// Brief: Slave Arm Adjust
FUNCTION_BLOCK PUBLIC FB_SlaveCtrlKineCaliSample EXTENDS FB_SlaveCtrlAdjust
VAR CONSTANT
	m_sampleNum :INT :=15;
END_VAR
VAR
	// sample joint position 
	m_sampleSetupJntPos :ARRAY[1..m_sampleNum] OF Vec5d;
	m_sampleSlaveJntPos :ARRAY[1..m_sampleNum] OF Vec6d;
	
	// sample signal
	m_sampleSignal : FB_AdjustLongPress;
	
	// current sample number
	m_curSampleNum :INT :=1;
	
	m_logStr:STRING;
	m_armStr:STRING;
	
END_VAR

// override this function in each exact controller
METHOD PROTECTED calcCmdJntPos : BOOL
VAR_IN_OUT CONSTANT
	i_endoscopePose : ST_Frame;
	i_masterStatus :ST_MasterStatus;
	i_setupStatus: ST_SetupStatus;
	i_slaveArm :FB_SlaveArm;
END_VAR
VAR
	i:INT;
END_VAR
SUPER^.calcCmdJntPos(i_endoscopePose,i_masterStatus, i_setupStatus, i_slaveArm);

IF m_curSampleNum > m_sampleNum THEN
	m_isFinished :=TRUE;
	AGILOG_DebugStop();
	RETURN;
END_IF
	
IF m_sampleSignal.run(i_slaveArm.m_adjustIO) THEN
	
	m_sampleSetupJntPos[m_curSampleNum] := SetupArmControl.m_setupRobot.m_setupArms[i_slaveArm.armIdx].curJntPos;
	m_sampleSlaveJntPos[m_curSampleNum] := i_slaveArm.curDHJntPos;
	
	AGILOG_DEBUG(m_armStr, FALSE, 1);
	
//	AGILOG_DEBUG(SetupArmControl.m_setupRobot.m_setupArms[i_slaveArm.armIdx].curJntPos, FALSE, 2);
//	AGILOG_DEBUG(i_slaveArm.curDHJntPos, FALSE, 1);
	
	AGILOG_DEBUG(RobotDynamics.m_instruViewCheck.m_instruPoseInScope[i_slaveArm.armIdx].m_pos,FALSE, 1);
	
	m_curSampleNum := m_curSampleNum +1;
END_IF
END_METHOD

METHOD PUBLIC Init : BOOL
VAR_IN_OUT CONSTANT
	i_slaveArm	:FB_SlaveArm;
END_VAR
VAR_IN_OUT 
	r_slaveArmCtrlCmd :ST_SlaveArmCtrlCmds;
END_VAR

VAR
	fileName:STRING;
END_VAR
//init
SUPER^.Init(i_slaveArm,r_slaveArmCtrlCmd);

m_curSampleNum:=1;
 
fileName := CONCAT('kineCaliSample_arm', INT_TO_STRING(i_slaveArm.armIdx));
fileName := CONCAT(fileName, '.txt');
AGILOG_DebugStart(fileName);

m_logStr := '########Start kinematic calibration sampling.########';
AGILOG_DEBUG(m_logStr, TRUE, 1);

m_armStr := concat('slaveArm', INT_TO_STRING(i_slaveArm.armIdx));
END_METHOD

END_FUNCTION_BLOCK

(* stored: Version 1.1.0.1, ProductVersion 3.1.4024.12
   POU FB_SlaveCtrlKineCaliSample: Id {02f01ec7-1d58-4e6b-a7e5-6da2475a150e}, SpecialFunc None
   Method calcCmdJntPos: Id {8eef563d-63aa-4579-9d6b-9b74bcf7e387}
   Method Init: Id {bbf7086f-25aa-4720-8f00-d9a234c6d91e} *)
